// TIA Portal V18 export
ORGANIZATION_BLOCK "12-Drive Unit"   // OB131, LAD, ProgramCycle
TITLE = "Main Program Sweep (Cycle)"
{ S7_Optimized_Access := 'TRUE' }
VERSION : 0.1
// stored: AutoNumber true, IsIECCheckEnabled false, SetENOAutomatically false
   VAR_INPUT
      Initial_Call : Bool;   // Initial call of this OB
      Remanence : Bool;   // =True, if remanent data are available
   END_VAR
   VAR_TEMP
      "Drive Angle NomScale" : Real;
      "Drive Left Slow Point" : Real;
      tempory0 : Byte;
      tempory1 : Byte;
      "Drive Compare OK" : Bool;
      "Drive Right Slow Point" : Real;
   END_VAR
BEGIN

REGION Network 1: Drive Unit Angle Sensor
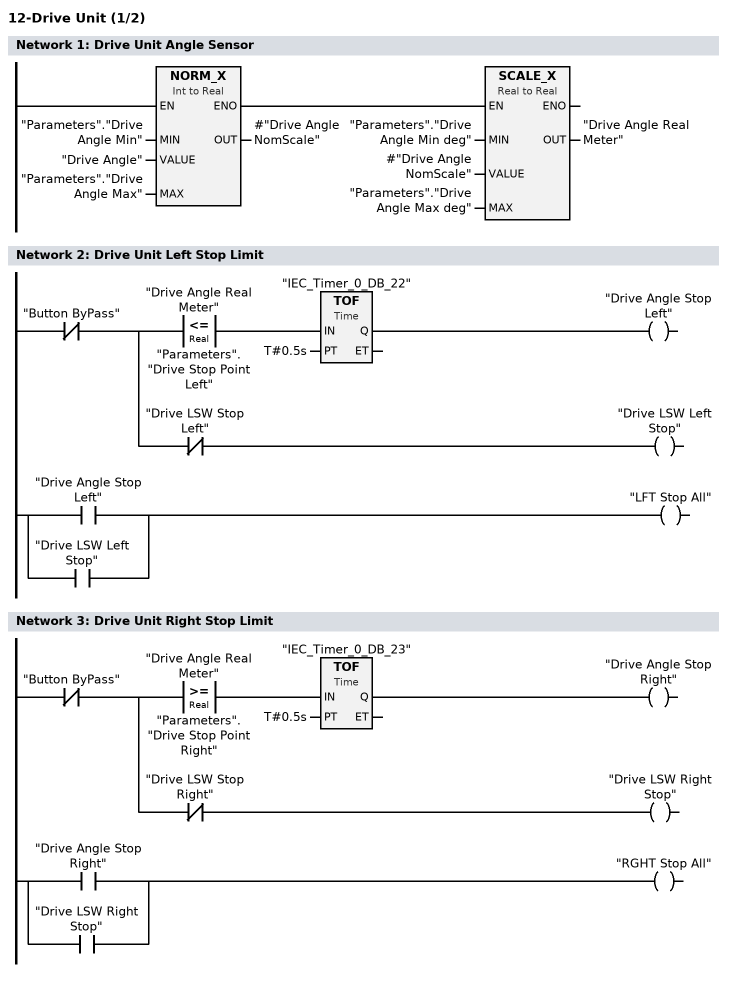
   RUNG wire#powerrail
      { S7_Templates := "[SrcType := Int, DestType := Real]" } Normalize(min := "Parameters"."Drive Angle Min", value := "Drive Angle", max := "Parameters"."Drive Angle Max", out => #"Drive Angle NomScale")
      { S7_Templates := "[SrcType := Real, DestType := Real]" } Scale(min := "Parameters"."Drive Angle Min deg", value := #"Drive Angle NomScale", max := "Parameters"."Drive Angle Max deg", out => "Drive Angle Real Meter")
   END_RUNG
   // the same network as SCL:
   #"Drive Angle NomScale" := NORM_X(MIN := "Parameters"."Drive Angle Min", VALUE := "Drive Angle", MAX := "Parameters"."Drive Angle Max");
   "Drive Angle Real Meter" := SCALE_X(MIN := "Parameters"."Drive Angle Min deg", VALUE := #"Drive Angle NomScale", MAX := "Parameters"."Drive Angle Max deg");
END_REGION

REGION Network 2: Drive Unit Left Stop Limit
   RUNG wire#powerrail
      I_Contact( "Button ByPass" )
      wire#w1
      { S7_Templates := "SrcType := Real" } LE_Contact(in1 := "Drive Angle Real Meter", in2 := "Parameters"."Drive Stop Point Left")
      { S7_Templates := "time_type := Time" } "IEC_Timer_0_DB_22".TOF(pt := T#0.5s, et =>)
      Coil( "Drive Angle Stop Left" )
   END_RUNG
   RUNG wire#w1
      I_Contact( "Drive LSW Stop Left" )
      Coil( "Drive LSW Left Stop" )
   END_RUNG
   RUNG wire#powerrail
      Contact( "Drive Angle Stop Left" )
      wire#w2
      Coil( "LFT Stop All" )
   END_RUNG
   RUNG wire#powerrail
      Contact( "Drive LSW Left Stop" )
   END_RUNG wire#w2
   // the same network as SCL:
   "IEC_Timer_0_DB_22".TOF(IN := NOT "Button ByPass" AND ("Drive Angle Real Meter" <= "Parameters"."Drive Stop Point Left"),
                           PT := T#0.5s);
   "Drive Angle Stop Left" := "IEC_Timer_0_DB_22".Q;
   "Drive LSW Left Stop" := NOT "Button ByPass" AND NOT "Drive LSW Stop Left";
   "LFT Stop All" := "Drive Angle Stop Left" OR "Drive LSW Left Stop";
END_REGION

REGION Network 3: Drive Unit Right Stop Limit
   RUNG wire#powerrail
      I_Contact( "Button ByPass" )
      wire#w1
      { S7_Templates := "SrcType := Real" } GE_Contact(in1 := "Drive Angle Real Meter", in2 := "Parameters"."Drive Stop Point Right")
      { S7_Templates := "time_type := Time" } "IEC_Timer_0_DB_23".TOF(pt := T#0.5s, et =>)
      Coil( "Drive Angle Stop Right" )
   END_RUNG
   RUNG wire#w1
      I_Contact( "Drive LSW Stop Right" )
      Coil( "Drive LSW Right Stop" )
   END_RUNG
   RUNG wire#powerrail
      Contact( "Drive Angle Stop Right" )
      wire#w2
      Coil( "RGHT Stop All" )
   END_RUNG
   RUNG wire#powerrail
      Contact( "Drive LSW Right Stop" )
   END_RUNG wire#w2
   // the same network as SCL:
   "IEC_Timer_0_DB_23".TOF(IN := NOT "Button ByPass" AND ("Drive Angle Real Meter" >= "Parameters"."Drive Stop Point Right"),
                           PT := T#0.5s);
   "Drive Angle Stop Right" := "IEC_Timer_0_DB_23".Q;
   "Drive LSW Right Stop" := NOT "Button ByPass" AND NOT "Drive LSW Stop Right";
   "RGHT Stop All" := "Drive Angle Stop Right" OR "Drive LSW Right Stop";
END_REGION

REGION Network 4: Drive Unit Slow Limits
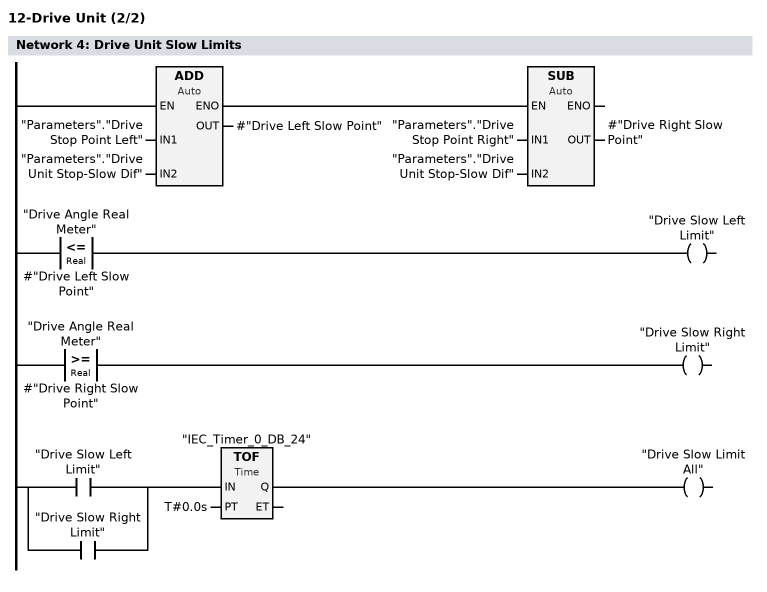
   RUNG wire#powerrail
      Add(in1 := "Parameters"."Drive Stop Point Left", in2 := "Parameters"."Drive Unit Stop-Slow Dif", out => #"Drive Left Slow Point")
      Sub(in1 := "Parameters"."Drive Stop Point Right", in2 := "Parameters"."Drive Unit Stop-Slow Dif", out => #"Drive Right Slow Point")
   END_RUNG
   RUNG wire#powerrail
      { S7_Templates := "SrcType := Real" } LE_Contact(in1 := "Drive Angle Real Meter", in2 := #"Drive Left Slow Point")
      Coil( "Drive Slow Left Limit" )
   END_RUNG
   RUNG wire#powerrail
      { S7_Templates := "SrcType := Real" } GE_Contact(in1 := "Drive Angle Real Meter", in2 := #"Drive Right Slow Point")
      Coil( "Drive Slow Right Limit" )
   END_RUNG
   RUNG wire#powerrail
      Contact( "Drive Slow Left Limit" )
      wire#w1
      { S7_Templates := "time_type := Time" } "IEC_Timer_0_DB_24".TOF(pt := T#0.0s, et =>)
      Coil( "Drive Slow Limit All" )
   END_RUNG
   RUNG wire#powerrail
      Contact( "Drive Slow Right Limit" )
   END_RUNG wire#w1
   // the same network as SCL:
   #"Drive Left Slow Point" := "Parameters"."Drive Stop Point Left" + "Parameters"."Drive Unit Stop-Slow Dif";
   #"Drive Right Slow Point" := "Parameters"."Drive Stop Point Right" - "Parameters"."Drive Unit Stop-Slow Dif";
   "Drive Slow Left Limit" := "Drive Angle Real Meter" <= #"Drive Left Slow Point";
   "Drive Slow Right Limit" := "Drive Angle Real Meter" >= #"Drive Right Slow Point";
   "IEC_Timer_0_DB_24".TOF(IN := "Drive Slow Left Limit" OR "Drive Slow Right Limit", PT := T#0.0s);
   "Drive Slow Limit All" := "IEC_Timer_0_DB_24".Q;
END_REGION
END_ORGANIZATION_BLOCK
